{attribute 'qualified_only'}
VAR_GLOBAL
    StartProcess : BOOL := FALSE;
    ResetProcess : BOOL := FALSE;

    AdsConnected : BOOL := FALSE;  // Node.js met TRUE si connect
END_VAR

(* stored: Version 1.1.0.1, ProductVersion 3.1.4024.0
   GVL GVL_Command: Id {12345678-1234-1234-1234-123456789004} *)
